(* PLC project cb_f_trig, Dassault Systèmes ControlBuild 2024x *)
(* stored: creationDateTime 2023-10-03T11:12:44-01:00 *)

(* This is a IEC 1131-3 falling edge *)
FUNCTION_BLOCK timers_counters.cb_f_trig
  VAR_INPUT
    IN : BOOL := false;
  END_VAR
  VAR_OUTPUT
    Q0 : BOOL := false;
  END_VAR
  VAR
    Mem : BOOL := false;
  END_VAR

(* --------------------------------------------------------------	*)
(* Type : BFU									*)
(* Copyright : Geensoft							*)
(* Version : 1.0 23/03/2010							*)
(* -------------------------------------------------------------	*)
(* This is a Falling Edge  (F_TRIG)					*)
(* -------------------------------------------------------------	*)

Q0 := not IN and  Mem;
Mem := IN;
END_FUNCTION_BLOCK
